FUNCTION_BLOCK ConfigManagerWidget
VAR_INPUT
END_VAR
VAR_OUTPUT
    actualStatus : StatusWidget;
    load : ReadXmlProcessWidget;
    save : WriteXmlProcessWidget;
END_VAR
VAR_IN_OUT
    mgr : ConfigManager;
END_VAR
VAR
END_VAR

actualStatus(
    text  := mgr.actualStatus,
    color := HealthBusyToColor(
        healthStatus := mgr.statuses.healthStatus,
        busyStatus := mgr.statuses.busyStatus));

load(process := mgr.processes.load);
save(process := mgr.processes.save);

END_FUNCTION_BLOCK

(* stored: Version 1.1.0.1, ProductVersion 3.1.4018.2
   POU ConfigManagerWidget: Id {6a8aba40-88af-4925-8ef4-d598e96c1c07}, SpecialFunc None *)
